Fanuc KAREL source: IO0104.KL

-- PROVISIONAL review KL for V940-1; original PC SHA256 1945e8d2881cbd6723b35efdaf5ab6717e85fa715180adadea89c7ce285cfa15
-- Incomplete behavior may be omitted. Consult companion uncertainty JSON. Do not deploy.
PROGRAM IO0104
%NOLOCKGROUP
-- UNRESOLVED_LOCAL_POOL 5 cells at code offset 13; source declarations unknown
-- DIRECT_LOCAL_WORD_ACCESS alone does not prove INTEGER, REAL, or BOOLEAN
BEGIN
  -- V9_ZERO_TABLE_METADATA_HINT layout=0001; no indexed target words; source/name/runtime held
  -- V9_ZERO_GLOBAL_LAYOUT_HINT count-one $GROUP table, zero relocation slots, two routine descriptors; executable preamble and source held
  -- V9_ANALOG_RDI_SIGNAL_HINT RDI read array_I
  -- UNRESOLVED_PC offsets 0-18; opcodes 2B,2C,7B
  -- UNRESOLVED_PC offsets 23-30; opcodes 9D,23
  -- UNRESOLVED_PC offsets 35-49; opcodes 2E,22,9D,33,35
  -- UNRESOLVED_PC offsets 54-61; opcodes 9D,23
  -- UNRESOLVED_PC offsets 66-77; opcodes 2E,23
  -- UNRESOLVED_PC offsets 82-104; opcodes 22,21,33,34,19,23
  -- UNRESOLVED_PC offsets 109-113; opcodes 7F
  -- UNRESOLVED_PC offsets 118-122; opcodes 27,AA
  -- UNRESOLVED_PC offsets 127-131; opcodes 7F
END IO0104
